(*
    This FB compares two instances of any object type and returns whether they
    are the same type, size and value or not. This is necessary for two reasons:
    1. So that we can know exactly what differs between the two input parameters
    2. It's not possible to do a comparison (= or <>) between two instances of ANY.
*)
FUNCTION_BLOCK FB_AnyComparator
VAR_INPUT
    AnyValueOne : ANY;
    AnyValueTwo : ANY;
END_VAR
VAR_OUTPUT
    DataTypesNotEquals : BOOL; // The data type of the two ANY input parameters are not equal
    DataSizeNotEquals : BOOL; // The data size of the two ANY input parameters are not equal
    DataContentNotEquals : BOOL; // The data content of the two ANY input parameters are not equal
END_VAR
VAR
    IteratorCounter : DINT;
END_VAR

(* Reset the outputs *)
DataTypesNotEquals := FALSE;
DataSizeNotEquals := FALSE;
DataContentNotEquals := FALSE;

(* Check whether the type of the inputs differs *)
IF AnyValueOne.TypeClass <> AnyValueTwo.TypeClass THEN
    DataTypesNotEquals := TRUE;
END_IF

(* Check whether the size of the inputs differs *)
IF NOT DataTypesNotEquals THEN
    IF (AnyValueOne.diSize <> AnyValueTwo.diSize) THEN
        DataSizeNotEquals := TRUE;
    END_IF
END_IF

(* Even though the data type and size are equals, the contents may still differ *)
IF NOT DataTypesNotEquals AND NOT DataSizeNotEquals THEN
    // Compare each byte in the ANY-types
    FOR IteratorCounter := 0 TO AnyValueOne.diSize - 1 BY 1 DO
        IF AnyValueOne.pValue[IteratorCounter] <> AnyValueTwo.pValue[IteratorCounter] THEN
            DataContentNotEquals := TRUE;
            EXIT;
        END_IF
    END_FOR
END_IF

END_FUNCTION_BLOCK

(* stored: Version 1.1.0.1, ProductVersion 3.1.4022.16
   POU FB_AnyComparator: Id {e4f95c0d-0ece-47a8-977f-f9d45a4f920e}, SpecialFunc None *)
